"C2GS1"	M 2318.0	BOOL	// (C2RB.S4): GRUPO DE SEQUENCIA PESO 1
"C2GS2"	M 2318.1	BOOL	// (C2RB.S4): GRUPO DE SEQUENCIA PESO 2
"C2GS4"	M 2318.2	BOOL	// (C2RB.S4): GRUPO DE SEQUENCIA PESO 4
"C2GS8"	M 2318.3	BOOL	// (C2RB.S4): GRUPO DE SEQUENCIA PESO 8
"C2E1_SRE"	M 2318.4	BOOL	// (C2RB.S4): INFO DETECCION RETROCESOSEQUENCIA 1
"C2E1_SAV"	M 2318.5	BOOL	// (C2RB.S4): INFO DETECCION AVANCE SEQUENCIA 1
"C2E2_SRE"	M 2318.6	BOOL	// (C2RB.S4): INFO DETECCION RETROCESOSEQUENCIA 2
"C2E2_SAV"	M 2318.7	BOOL	// (C2RB.S4): INFO DETECCION AVANCE SEQUENCIA 2
"C2DECH"	M 2319.0	BOOL	// (C2RB.S4): COMANDE DESBLOQUEIO TROCADER
"C2EVO1"	M 2320.0	BOOL	// (C2RB.S5): EVENTO HERRAMIENTA 1
"C2EVO2"	M 2320.1	BOOL	// (C2RB.S5): EVENTO HERRAMIENTA 2
"C2EVO3"	M 2320.2	BOOL	// (C2RB.S5): EVENTO HERRAMIENTA 3
"C2EVO4"	M 2320.3	BOOL	// (C2RB.S5): EVENTO HERRAMIENTA 4
"C2EVO5"	M 2320.4	BOOL	// (C2RB.S5): EVENTO HERRAMIENTA 5
"C2EVO6"	M 2320.5	BOOL	// (C2RB.S5): EVENTO HERRAMIENTA 6
"C2EVO7"	M 2320.6	BOOL	// (C2RB.S5): EVENTO HERRAMIENTA 7
"C2EVO8"	M 2320.7	BOOL	// (C2RB.S5): EVENTO HERRAMIENTA 8
"C2EVO9"	M 2321.0	BOOL	// (C2RB.S5): EVENTO HERRAMIENTA 9
"C2EVO10"	M 2321.1	BOOL	// (C2RB.S5): EVENTO HERRAMIENTA 10
"C2EVO11"	M 2321.2	BOOL	// (C2RB.S5): EVENTO HERRAMIENTA 11
"C2EVO12"	M 2321.3	BOOL	// (C2RB.S5): EVENTO HERRAMIENTA 12
"C2EVO13"	M 2321.4	BOOL	// (C2RB.S5): EVENTO HERRAMIENTA 13
"C2EVO14"	M 2321.5	BOOL	// (C2RB.S5): EVENTO HERRAMIENTA 14
"C2EVO15"	M 2321.6	BOOL	// (C2RB.S5): EVENTO HERRAMIENTA 15
"C2EVO16"	M 2321.7	BOOL	// (C2RB.S5): EVENTO HERRAMIENTA 16
"C2EV17"	M 2326.0	BOOL	// (C2RB.S8): EVENTO 17
"C2EV18"	M 2326.1	BOOL	// (C2RB.S8): EVENTO 18
"C2EV19"	M 2326.2	BOOL	// (C2RB.S8): EVENTO 19
"C2EV20"	M 2326.3	BOOL	// (C2RB.S8): EVENTO 20
"C2EV21"	M 2326.4	BOOL	// (C2RB.S8): EVENTO 21
"C2EV22"	M 2326.5	BOOL	// (C2RB.S8): EVENTO 22
"C2EV23"	M 2326.6	BOOL	// (C2RB.S8): EVENTO 23
"C2EV24"	M 2326.7	BOOL	// (C2RB.S8): EVENTO 24
"C2EV25"	M 2327.0	BOOL	// (C2RB.S8): EVENTO 25
"C2EV26"	M 2327.1	BOOL	// (C2RB.S8): EVENTO 26
"C2EV27"	M 2327.2	BOOL	// (C2RB.S8): EVENTO 27
"C2EV28"	M 2327.3	BOOL	// (C2RB.S8): EVENTO 28
"C2EV29"	M 2327.4	BOOL	// (C2RB.S8): EVENTO 29
"C2EV30"	M 2327.5	BOOL	// (C2RB.S8): EVENTO 30
"C2EV31"	M 2327.6	BOOL	// (C2RB.S8): EVENTO 31
"C2EV32"	M 2327.7	BOOL	// (C2RB.S8): EVENTO 32
"A2RBMS1_P"	MB 2200	BYTE	// BYTE 1 GENERAL DATA / GENERALITES
"A2RBMS2_P"	MB 2201	BYTE	// BYTE 2 GENERAL DATA / GENERALITES
"A2RBMS3_P"	MB 2202	BYTE	// BYTE 3 ROBOTT ORDERS / ORDRES ROBOTT
"A2RBMS4_P"	MB 2203	BYTE	// BYTE 4 ROBOTT ORDERS / ORDRES ROBOTT
"A2RBMS5_P"	MB 2204	BYTE	// BYTE 5 GRIPPER AND TOOL CHANGER / PREHENSEUR ET CHANGEUR OUTIL
"A2RBMS6_P"	MB 2205	BYTE	// BYTE 6 GRIPPER AND TOOL CHANGER / PREHENSEUR ET CHANGEUR OUTIL
"A2RBMS7_P"	MB 2206	BYTE	// BYTE 7 FAULT NUMBER / NUMERO DE DEFAUT
"A2RBMS8_P"	MB 2207	BYTE	// BYTE 8 FAULT NUMBER / NUMERO DE DEFAUT
"A2RBMS9_P"	MB 2208	BYTE	// BYTE 9 TOOL ORDERS/ ORDRES OUTIL
"A2RBMS10_P"	MB 2209	BYTE	// BYTE 10 TOOL ORDERS/ ORDRES OUTIL
"A2RBMS11_P"	MB 2210	BYTE	// BYTE 11
"A2RBMS12_P"	MB 2211	BYTE	// BYTE 12
"A2RBMS13_P"	MB 2212	BYTE	// BYTE 13
"A2RBMS14_P"	MB 2213	BYTE	// BYTE 14
"A2RBMS15_P"	MB 2214	BYTE	// BYTE 15
"A2RBMS16_P"	MB 2215	BYTE	// BYTE 16
"A2RBME1_P"	MB 2216	BYTE	// BYTE 1 GENERAL DATA AND CYCLE CODE / CODE CYCLE ET GENERALITES
"A2RBME2_P"	MB 2217	BYTE	// BYTE 2 GENERAL DATA AND CYCLE CODE / CODE CYCLE ET GENERALITES
"A2RBME3_P"	MB 2218	BYTE	// BYTE 3 ROBOTT EVENTS / EVENTOS ROBOTT
"A2RBME4_P"	MB 2219	BYTE	// BYTE 4 ROBOTT EVENTS / EVENTOS ROBOTT
"A2RBME5_P"	MB 2220	BYTE	// BYTE 5 GENERAL DATAS / GENERALITES
"A2RBME6_P"	MB 2221	BYTE	// BYTE 6 GENERAL DATAS / GENERALITES
"A2RBME7_P"	MB 2222	BYTE	// BYTE 7 GRIPPER AND TOOL CHANGER / PREHENSEUR ET CHANGEUR OUTIL
"A2RBME8_P"	MB 2223	BYTE	// BYTE 8 GRIPPER AND TOOL CHANGER / PREHENSEUR ET CHANGEUR OUTIL
"A2RBME9_P"	MB 2224	BYTE	// BYTE 9 TOOL EVENTS / EVENTOS OUTIL
"A2RBME10_P"	MB 2225	BYTE	// BYTE 10 TOOL EVENTS / EVENTOS OUTIL
"A2RBME11_P"	MB 2226	BYTE	// BYTE 11
"A2RBME12_P"	MB 2227	BYTE	// BYTE 12
"A2RBME13_P"	MB 2228	BYTE	// BYTE 13
"A2RBME14_P"	MB 2229	BYTE	// BYTE 14
"A2RBME15_P"	MB 2230	BYTE	// BYTE 15
"A2RBME16_P"	MB 2231	BYTE	// BYTE 16
"A3RBMS1_P"	MB 2232	BYTE	// BYTE 1 GENERAL DATA / GENERALITES
"A3RBMS2_P"	MB 2233	BYTE	// BYTE 2 GENERAL DATA / GENERALITES
"A3RBMS3_P"	MB 2234	BYTE	// BYTE 3 ROBOTT ORDERS / ORDRES ROBOTT
"A3RBMS4_P"	MB 2235	BYTE	// BYTE 4 ROBOTT ORDERS / ORDRES ROBOTT
"A3RBMS5_P"	MB 2236	BYTE	// BYTE 5 GRIPPER AND TOOL CHANGER / PREHENSEUR ET CHANGEUR OUTIL
"A3RBMS6_P"	MB 2237	BYTE	// BYTE 6 GRIPPER AND TOOL CHANGER / PREHENSEUR ET CHANGEUR OUTIL
"A3RBMS7_P"	MB 2238	BYTE	// BYTE 7 FAULT NUMBER / NUMERO DE DEFAUT
"A3RBMS8_P"	MB 2239	BYTE	// BYTE 8 FAULT NUMBER / NUMERO DE DEFAUT
"A3RBMS9_P"	MB 2240	BYTE	// BYTE 9 TOOL ORDERS/ ORDRES OUTIL
"A3RBMS10_P"	MB 2241	BYTE	// BYTE 10 TOOL ORDERS/ ORDRES OUTIL
"A3RBMS11_P"	MB 2242	BYTE	// BYTE 11
"A3RBMS12_P"	MB 2243	BYTE	// BYTE 12
"A3RBMS13_P"	MB 2244	BYTE	// BYTE 13
"A3RBMS14_P"	MB 2245	BYTE	// BYTE 14
"A3RBMS15_P"	MB 2246	BYTE	// BYTE 15
"A3RBMS16_P"	MB 2247	BYTE	// BYTE 16
"A3RBME1_P"	MB 2248	BYTE	// BYTE 1 GENERAL DATA AND CYCLE CODE / CODE CYCLE ET GENERALITES
"A3RBME2_P"	MB 2249	BYTE	// BYTE 2 GENERAL DATA AND CYCLE CODE / CODE CYCLE ET GENERALITES
"A3RBME3_P"	MB 2250	BYTE	// BYTE 3 ROBOTT EVENTS / EVENTOS ROBOTT
"A3RBME4_P"	MB 2251	BYTE	// BYTE 4 ROBOTT EVENTS / EVENTOS ROBOTT
"A3RBME5_P"	MB 2252	BYTE	// BYTE 5 GENERAL DATAS / GENERALITES
"A3RBME6_P"	MB 2253	BYTE	// BYTE 6 GENERAL DATAS / GENERALITES
"A3RBME7_P"	MB 2254	BYTE	// BYTE 7 GRIPPER AND TOOL CHANGER / PREHENSEUR ET CHANGEUR OUTIL
"A3RBME8_P"	MB 2255	BYTE	// BYTE 8 GRIPPER AND TOOL CHANGER / PREHENSEUR ET CHANGEUR OUTIL
"A3RBME9_P"	MB 2256	BYTE	// BYTE 9 TOOL EVENTS / EVENTOS OUTIL
"A3RBME10_P"	MB 2257	BYTE	// BYTE 10 TOOL EVENTS / EVENTOS OUTIL
"A3RBME11_P"	MB 2258	BYTE	// BYTE 11
"A3RBME12_P"	MB 2259	BYTE	// BYTE 12
"A3RBME13_P"	MB 2260	BYTE	// BYTE 13
"A3RBME14_P"	MB 2261	BYTE	// BYTE 14
"A3RBME15_P"	MB 2262	BYTE	// BYTE 15
"A3RBME16_P"	MB 2263	BYTE	// BYTE 16
"C2RBMS1_P"	MB 2296	BYTE	// BYTE 1 GENERAL DATA / GENERALITES
"C2RBMS2_P"	MB 2297	BYTE	// BYTE 2 GENERAL DATA / GENERALITES
"C2RBMS3_P"	MB 2298	BYTE	// BYTE 3 ROBOTT ORDERS / ORDRES ROBOTT
"C2RBMS4_P"	MB 2299	BYTE	// BYTE 4 ROBOTT ORDERS / ORDRES ROBOTT
"C2RBMS5_P"	MB 2300	BYTE	// BYTE 5 GRIPPER AND TOOL CHANGER / PREHENSEUR ET CHANGEUR OUTIL
"C2RBMS6_P"	MB 2301	BYTE	// BYTE 6 GRIPPER AND TOOL CHANGER / PREHENSEUR ET CHANGEUR OUTIL
"C2RBMS7_P"	MB 2302	BYTE	// BYTE 7 FAULT NUMBER / NUMERO DE DEFAUT
"C2RBMS8_P"	MB 2303	BYTE	// BYTE 8 FAULT NUMBER / NUMERO DE DEFAUT
"C2RBMS9_P"	MB 2304	BYTE	// BYTE 9 TOOL ORDERS/ ORDRES OUTIL
"C2RBMS10_P"	MB 2305	BYTE	// BYTE 10 TOOL ORDERS/ ORDRES OUTIL
"C2RBMS11_P"	MB 2306	BYTE	// BYTE 11
"C2RBMS12_P"	MB 2307	BYTE	// BYTE 12
"C2RBMS13_P"	MB 2308	BYTE	// BYTE 13
"C2RBMS14_P"	MB 2309	BYTE	// BYTE 14
"C2RBMS15_P"	MB 2310	BYTE	// BYTE 15
"C2RBMS16_P"	MB 2311	BYTE	// BYTE 16
"C2RBME1_P"	MB 2312	BYTE	// BYTE 1 GENERAL DATA AND CYCLE CODE / CODE CYCLE ET GENERALITES
"C2RBME2_P"	MB 2313	BYTE	// BYTE 2 GENERAL DATA AND CYCLE CODE / CODE CYCLE ET GENERALITES
"C2RBME3_P"	MB 2314	BYTE	// BYTE 3 ROBOTT EVENTS / EVENTOS ROBOTT
"C2RBME4_P"	MB 2315	BYTE	// BYTE 4 ROBOTT EVENTS / EVENTOS ROBOTT
"C2RBME5_P"	MB 2316	BYTE	// BYTE 5 GENERAL DATAS / GENERALITES
"C2RBME6_P"	MB 2317	BYTE	// BYTE 6 GENERAL DATAS / GENERALITES
"C2RBME7_P"	MB 2318	BYTE	// BYTE 7 GRIPPER AND TOOL CHANGER / PREHENSEUR ET CHANGEUR OUTIL
"C2RBME8_P"	MB 2319	BYTE	// BYTE 8 GRIPPER AND TOOL CHANGER / PREHENSEUR ET CHANGEUR OUTIL
"C2RBME9_P"	MB 2320	BYTE	// BYTE 9 TOOL EVENTS / EVENTOS OUTIL
"C2RBME10_P"	MB 2321	BYTE	// BYTE 10 TOOL EVENTS / EVENTOS OUTIL
"C2RBME11_P"	MB 2322	BYTE	// BYTE 11
"C2RBME12_P"	MB 2323	BYTE	// BYTE 12
"C2RBME13_P"	MB 2324	BYTE	// BYTE 13
"C2RBME14_P"	MB 2325	BYTE	// BYTE 14
"C2RBME15_P"	MB 2326	BYTE	// BYTE 15
"C2RBME16_P"	MB 2327	BYTE	// BYTE 16
"A2RBMS1_W"	MW 2200	WORD	// WORD 1 GENERAL DATA / GENERALITES
"A2RBMS2_W"	MW 2202	WORD	// WORD 2 ROBOTT ORDERS / ORDRES ROBOTT
"A2RBMS3_W"	MW 2204	WORD	// WORD 3 GRIPPER AND TOOL CHANGER / PREHENSEUR ET CHANGEUR OUTIL
"A2RBMS4_W"	MW 2206	WORD	// WORD 4 FAULT NUMBER / NUMERO DE DEFAUT
"A2RBMS5_W"	MW 2208	WORD	// WORD 5 TOOL ORDERS/ ORDRES OUTIL
"A2RBMS6_W"	MW 2210	WORD	// WORD 6
"A2RBMS7_W"	MW 2212	WORD	// WORD 7
"A2RBMS8_W"	MW 2214	WORD	// WORD 8
"A2RBME1_W"	MW 2216	WORD	// WORD 1 GENERAL DATA AND CYCLE CODE / CODE CYCLE ET GENERALITES
"A2RBME2_W"	MW 2218	WORD	// WORD 2 ROBOTT EVENTS / EVENTOS ROBOTT
"A2RBME3_W"	MW 2220	WORD	// WORD 3 GENERAL DATAS / GENERALITES
"A2RBME4_W"	MW 2222	WORD	// WORD 4 GRIPPER AND TOOL CHANGER / PREHENSEUR ET CHANGEUR OUTIL
"A2RBME5_W"	MW 2224	WORD	// WORD 5 TOOL EVENTS / EVENTOS OUTIL
"A2RBME6_W"	MW 2226	WORD	// WORD 6
"A2RBME7_W"	MW 2228	WORD	// WORD 7
"A2RBME8_W"	MW 2230	WORD	// WORD 8
"A3RBMS1_W"	MW 2232	WORD	// WORD 1 GENERAL DATA / GENERALITES
"A3RBMS2_W"	MW 2234	WORD	// WORD 2 ROBOTT ORDERS / ORDRES ROBOTT
"A3RBMS3_W"	MW 2236	WORD	// WORD 3 GRIPPER AND TOOL CHANGER / PREHENSEUR ET CHANGEUR OUTIL
"A3RBMS4_W"	MW 2238	WORD	// WORD 4 FAULT NUMWER / NUMERO DE DEFAUT
"A3RBMS5_W"	MW 2240	WORD	// WORD 5 TOOL ORDERS/ ORDRES OUTIL
"A3RBMS6_W"	MW 2242	WORD	// WORD 6
"A3RBMS7_W"	MW 2244	WORD	// WORD 7
"A3RBMS8_W"	MW 2246	WORD	// WORD 8
"A3RBME1_W"	MW 2248	WORD	// WORD 1 GENERAL DATA AND CYCLE CODE / CODE CYCLE ET GENERALITES
"A3RBME2_W"	MW 2250	WORD	// WORD 2 ROBOTT EVENTS / EVENTOS ROBOTT
"A3RBME3_W"	MW 2252	WORD	// WORD 3 GENERAL DATAS / GENERALITES
"A3RBME4_W"	MW 2254	WORD	// WORD 4 GRIPPER AND TOOL CHANGER / PREHENSEUR ET CHANGEUR OUTIL
"A3RBME5_W"	MW 2256	WORD	// WORD 5 TOOL EVENTS / EVENTOS OUTIL
"A3RBME6_W"	MW 2258	WORD	// WORD 6
"A3RBME7_W"	MW 2260	WORD	// WORD 7
"A3RBME8_W"	MW 2262	WORD	// WORD 8
"C2RBMS1_W"	MW 2296	WORD	// WORD 1 GENERAL DATA / GENERALITES
"C2RBMS2_W"	MW 2298	WORD	// WORD 2 ROBOTT ORDERS / ORDRES ROBOTT
"C2RBMS3_W"	MW 2300	WORD	// WORD 3 GRIPPER AND TOOL CHANGER / PREHENSEUR ET CHANGEUR OUTIL
"C2RBMS4_W"	MW 2302	WORD	// WORD 4 FAULT NUMWER / NUMERO DE DEFAUT
"C2RBMS5_W"	MW 2304	WORD	// WORD 5 TOOL ORDERS/ ORDRES OUTIL
"C2RBMS6_W"	MW 2306	WORD	// WORD 6
"C2RBMS7_W"	MW 2308	WORD	// WORD 7
"C2RBMS8_W"	MW 2310	WORD	// WORD 8
"C2RBME1_W"	MW 2312	WORD	// WORD 1 GENERAL DATA AND CYCLE CODE / CODE CYCLE ET GENERALITES
"C2RBME2_W"	MW 2314	WORD	// WORD 2 ROBOTT EVENTS / EVENTOS ROBOTT
"C2RBME3_W"	MW 2316	WORD	// WORD 3 GENERAL DATAS / GENERALITES
"C2RBME4_W"	MW 2318	WORD	// WORD 4 GRIPPER AND TOOL CHANGER / PREHENSEUR ET CHANGEUR OUTIL
"C2RBME5_W"	MW 2320	WORD	// WORD 5 TOOL EVENTS / EVENTOS OUTIL
"C2RBME6_W"	MW 2322	WORD	// WORD 6
"C2RBME7_W"	MW 2324	WORD	// WORD 7
"C2RBME8_W"	MW 2326	WORD	// WORD 8
"CYCL_EXC"	OB 1	OB 1	// EXECUTION CYCLE
"CYC_INT4"	OB 34	OB 34	// CYCLIC INTERRUPT 4
"CYCL_FLT"	OB 80	OB 80	// Cycle Time Fault
"I/O_FLT1"	OB 82	OB 82	// I/O POINT FAULT 1
"I/O_FLT2"	OB 83	OB 83	// I/O POINT FAULT 2
"OBNL_FLT"	OB 85	OB 85	// OB NOT LOADED FAULT
"RACK_FLT"	OB 86	OB 86	// LOSS OF RACK FAULT
"COMPLETE RESTART"	OB 100	OB 100	// COMPLETE RESTART
"PROG_ERR"	OB 121	OB 121	// Programming Error
"MOD_ERR"	OB 122	OB 122	// MODULE ACCESS ERROR
"VADI"	Q 0.0	BOOL	// (MOP-IM.M06-07): INDICDOR RESET FALLA
"VMCY"	Q 0.1	BOOL	// (MOP-IM.M06-07): INDICADOR MARCHA CICLO
"VAOP"	Q 0.3	BOOL	// (MOP-IM.M06-07): ALIMENTADOR APPEL OPERADOR
"Z1VROC"	Q 10.0	BOOL	// (Z1ZB.M05): INDICADOR Retorno Origen
"Z1RCM"	Q 10.7	BOOL	// (Z1ZB.M05): RELE DE CONTROL DE MASA
"RAU"	Q 25.0	BOOL	// (Z1ZB.M15): RELE COMUN DE SEGURIDAD SC1 (Z1AU)
"RES"	Q 25.1	BOOL	// (Z1ZB.M15): RELE COMUN DE SEGURIDAD ES
"RFZ"	Q 25.2	BOOL	// (Z1ZB.M15): RELE COMUN DE SEGURIDAD FZ
"RSC4"	Q 25.3	BOOL	// (Z1ZB.M15): RELE COMUN DE SEGURIDAD RL
"WB11"	Q 42.0	BOOL	// (Z1ZB.M08):Welding Box 1 Bit 1
"WB12"	Q 42.1	BOOL	// (Z1ZB.M08):Welding Box 1 Bit 2
"WB13"	Q 42.2	BOOL	// (Z1ZB.M08):Welding Box 1 Bit 3
"WB14"	Q 42.3	BOOL	// (Z1ZB.M08):Welding Box 1 Bit 4
"WB21"	Q 42.4	BOOL	// (Z1ZB.M08):Welding Box 2 Bit 1
"WB22"	Q 42.5	BOOL	// (Z1ZB.M08):Welding Box 2 Bit 2
"WB23"	Q 42.6	BOOL	// (Z1ZB.M08):Welding Box 2 Bit 3
"WB24"	Q 42.7	BOOL	// (Z1ZB.M08):Welding Box 2 Bit 4
"OP1VAT"	Q 43.0	BOOL	// (Z1ZB.M09): Work Autorisation Lamp 1 (Green)
"OP1VIT"	Q 43.1	BOOL	// (Z1ZB.M09): Work Prohibition Lamp 1 (Red)
"OP1VDF"	Q 43.2	BOOL	// (Z1ZB.M09): Default Lamp 1 (Orange)
"A0CBNOK"	Q 43.3	BOOL	// (Z1ZB.M09): BARCODE READING NOK
"A0CBOK"	Q 43.4	BOOL	// (Z1ZB.M09): BARCODE READING OK
"OP2VAT"	Q 43.5	BOOL	// (Z1ZB.M09): Work Autorisation Lamp 2 (Green)
"OP2VIT"	Q 43.6	BOOL	// (Z1ZB.M09): Work Prohibition Lamp 2 (Red)
"OP2VDF"	Q 43.7	BOOL	// (Z1ZB.M09): Default Lamp 2 (Orange)
"A0EACH1"	Q 60.0	BOOL	// ELECTROVALVE AV CH1
"A0ERCH1"	Q 60.1	BOOL	// ELECTROVALVE RET CH1
"A0EAVR2"	Q 60.2	BOOL	// ELECTROVALVE AV VR2
"A0ERVR2"	Q 60.3	BOOL	// ELECTROVALVE RET VR2
"A0EAVR3"	Q 60.4	BOOL	// ELECTROVALVE AV VR3
"A0ERVR3"	Q 60.5	BOOL	// ELECTROVALVE RET VR3
"A0EASR4"	Q 60.6	BOOL	// ELECTROVALVE AV SR4
"A0ERSR4"	Q 60.7	BOOL	// ELECTROVALVE RET SR4
"A0EASR5"	Q 61.0	BOOL	// ELECTROVALVE AV SR5
"A0ERSR5"	Q 61.1	BOOL	// ELECTROVALVE RET SR5
"A0EASR6"	Q 61.2	BOOL	// ELECTROVALVE AV SR6
"A0ERSR6"	Q 61.3	BOOL	// ELECTROVALVE RET SR6
"A0EASR7"	Q 61.4	BOOL	// ELECTROVALVE AV SR7
"A0ERSR7"	Q 61.5	BOOL	// ELECTROVALVE RET SR7
"A0EASR9"	Q 62.0	BOOL	// ELECTROVALVE AV SR9
"A0ERSR9"	Q 62.1	BOOL	// ELECTROVALVE RET SR9
"A0RSOP"	Q 68.0	BOOL	// (A0IM1-FVD0): SEG OPERADOR
"A0EV"	Q 68.2	BOOL	// (A0IM1-FVD0): PILOTAGE ELETROVALVE (COMMON ES)
"A0_DO8"	Q 259.0	BOOL	// (A0SBS120): DIGITAL OUTPUT 8
"A0_DO9"	Q 259.1	BOOL	// (A0SBS120): DIGITAL OUTPUT 9
"A0_DO10"	Q 259.2	BOOL	// (A0SBS120): DIGITAL OUTPUT 10
"A0_DO11"	Q 259.3	BOOL	// (A0SBS120): DIGITAL OUTPUT 11
"A0_STO_O"	Q 312.0	BOOL	// (A0SBS120): ENABLE STO
"A0_SS1_O"	Q 312.1	BOOL	// (A0SBS120): ENABLE SS1
"A0_SS2_O"	Q 312.2	BOOL	// (A0SBS120): ENABLE SS2
"A0_SOS_O"	Q 312.3	BOOL	// (A0SBS120): ENABLE SOS
"A0_SLS_O"	Q 312.4	BOOL	// (A0SBS120): ENABLE SLS
"A0_RES1_O"	Q 312.5	BOOL	// (A0SBS120): RESERVE
"A0_RES2_O"	Q 312.6	BOOL	// (A0SBS120): RESERVE
"A0_ACK_O"	Q 312.7	BOOL	// (A0SBS120): ACK
"A0_RES3_O"	Q 313.0	BOOL	// (A0SBS120): RESERVE
"A0_L1SLS_O"	Q 313.1	BOOL	// (A0SBS120): ENABLE LIMIT 1 SLS
"A0_L2SLS_O"	Q 313.2	BOOL	// (A0SBS120): ENABLE LIMIT 2 SLS
"A0_RES4_O"	Q 313.3	BOOL	// (A0SBS120): RESERVE
"A0_RES5_O"	Q 313.4	BOOL	// (A0SBS120): RESERVE
"A0_RES6_O"	Q 313.5	BOOL	// (A0SBS120): RESERVE
"A0_RES7_O"	Q 313.6	BOOL	// (A0SBS120): RESERVE
"A0_RES8_O"	Q 313.7	BOOL	// (A0SBS120): RESERVE
"Z1SPA1VMCY"	Q 350.7	BOOL	// (Z1SPA1.O0): INDICADOR MARCHA CICLO
"Z1SPA1VDACY"	Q 351.0	BOOL	// (Z1SPA1.O1): INDICADOR DEMANDA PARADA CICLO
"Z2VROC"	Q 400.0	BOOL	// (Z2ZB.M07): INDICADOR Retorno Origen
"Z2VMCY"	Q 400.1	BOOL	// Z2ZB[M07]: LAMP CYCLE RUN (SOP)
"Z2RCM"	Q 400.7	BOOL	// (Z2ZB.M07): RELE DE CONTROL DE MASA
"B0WB11"	Q 401.0	BOOL	// (Z2ZB.M08):Welding Box 1 Bit 1
"B0WB12"	Q 401.1	BOOL	// (Z2ZB.M08):Welding Box 1 Bit 2
"B0WB13"	Q 401.2	BOOL	// (Z2ZB.M08):Welding Box 1 Bit 3
"B0WB14"	Q 401.3	BOOL	// (Z2ZB.M08):Welding Box 1 Bit 4
"B0WB21"	Q 401.4	BOOL	// (Z2ZB.M08):Welding Box 2 Bit 1
"B0WB22"	Q 401.5	BOOL	// (Z2ZB.M08):Welding Box 2 Bit 2
"B0WB23"	Q 401.6	BOOL	// (Z2ZB.M08):Welding Box 2 Bit 3
"B0WB24"	Q 401.7	BOOL	// (Z2ZB.M08):Welding Box 2 Bit 4
"B0OP1VAT"	Q 402.0	BOOL	// (Z2ZB.M08): Work Autorisation Lamp 1 (Green)
"B0OP1VIT"	Q 402.1	BOOL	// (Z2ZB.M08): Work Prohibition Lamp 1 (Red)
"B0OP1VDF"	Q 402.2	BOOL	// (Z2ZB.M08): Default Lamp 1 (Orange)
"A402.3"	Q 402.3	BOOL	// (Z2ZB.M08): RESERVE
"A402.4"	Q 402.4	BOOL	// (Z2ZB.M08): RESERVE
"B0OP2VAT"	Q 402.5	BOOL	// (Z2ZB.M08): Work Autorisation Lamp 2 (Green)
"B0OP2VIT"	Q 402.6	BOOL	// (Z2ZB.M08): Work Prohibition Lamp 2 (Red)
"B0OP2VDF"	Q 402.7	BOOL	// (Z2ZB.M08): Default Lamp 2 (Orange)
"B0RAU"	Q 423.0	BOOL	// (Z2ZB.M13): RELE COMUN DE SEGURIDAD SC1 (Z2AU)
"B0RES"	Q 423.1	BOOL	// (Z2ZB.M13): RELE COMUN DE SEGURIDAD ES
"B0RFZ"	Q 423.2	BOOL	// (Z2ZB.M13): RELE COMUN DE SEGURIDAD FZ
"B0RSC4"	Q 423.3	BOOL	// (Z2ZB.M13): RELE COMUN DE SOP
"B0EASR1"	Q 450.0	BOOL	// ELECTROVALVE AV SR1
"B0ERSR1"	Q 450.1	BOOL	// ELECTROVALVE RET SR1
"B0EASR2"	Q 450.2	BOOL	// ELECTROVALVE AV SR2
"B0ERSR2"	Q 450.3	BOOL	// ELECTROVALVE RET SR2
"B0EASR3"	Q 450.4	BOOL	// ELECTROVALVE AV SR3
"B0ERSR3"	Q 450.5	BOOL	// ELECTROVALVE RET SR3
"B0EASR4"	Q 450.6	BOOL	// ELECTROVALVE AV SR4
"B0ERSR4"	Q 450.7	BOOL	// ELECTROVALVE RET SR4
"B0EASR5"	Q 451.0	BOOL	// ELECTROVALVE AV SR5
"B0ERSR5"	Q 451.1	BOOL	// ELECTROVALVE RET SR5
"B0EASR6"	Q 451.2	BOOL	// ELECTROVALVE AV SR6
"B0ERSR6"	Q 451.3	BOOL	// ELECTROVALVE RET SR6
"B0EASR7"	Q 451.4	BOOL	// ELECTROVALVE AV SR7
"B0ERSR7"	Q 451.5	BOOL	// ELECTROVALVE RET SR7
"B0EASR8"	Q 451.6	BOOL	// ELECTROVALVE AV SR8
"B0ERSR8"	Q 451.7	BOOL	// ELECTROVALVE RET SR8
"B0EACL9"	Q 452.0	BOOL	// ELECTROVALVE AV CL9
"B0ERCL9"	Q 452.1	BOOL	// ELECTROVALVE RET CL9
"B0EACL10"	Q 452.2	BOOL	// ELECTROVALVE AV CL10
"B0ERCL10"	Q 452.3	BOOL	// ELECTROVALVE RET CL10
"RES1"	Q 452.4	BOOL
"RES2"	Q 452.5	BOOL
"RES3"	Q 452.6	BOOL
"RES4"	Q 452.7	BOOL
"Z2SPA1VMCY"	Q 490.7	BOOL	// (Z2SPA1.O0): INDICADOR MARCHA CICLO
"Z2SPA1VDACY"	Q 491.0	BOOL	// (Z2SPA1.O1): INDICADOR DEMANDA PARADA CICLO
"BOSEW_POS_ESCRITA"	QW 434	WORD
"TP"	SFB 3	SFB 3	// GENERATE A PULSE
"TON"	SFB 4	SFB 4	// GENERATE AN ON DELAY
"TOF"	SFB 5	SFB 5	// GENERATE AN OFF DELAY
"RDREC"	SFB 52	SFB 52	// READ A PROCESS DATA RECORD
"WRREC"	SFB 53	SFB 53	// WRITE A PROCESS DATA RECORD
"RALRM"	SFB 54	SFB 54	// Receive Alarm Data
"SET_CLK"	SFC 0	SFC 0	// SET SYSTEM CLOCK
"READ_CLK"	SFC 1	SFC 1	// READ SYSTEM CLOCK
"RD_SINFO"	SFC 6	SFC 6	// READ OB START INFORMATION
"D_ACT_DP"	SFC 12	SFC 12	// DEACTIVATING AND ACTIVATING DP SLAVES
"DPRD_DAT"	SFC 14	SFC 14	// READ CONSISTENT DATA OF A STANDARD DP SLAVE
"DPWR_DAT"	SFC 15	SFC 15	// WRITE CONSISTENT DATA TO A STANDARD DP SLAVE
"ALARM_SQ"	SFC 17	SFC 17	// Generate Block-Related Messages with Acknowledgment
"BLKMOV"	SFC 20	SFC 20	// COPY VARIABLES
"FILL"	SFC 21	SFC 21	// INITIALIZE A MEMORY AREA
"TEST_DB"	SFC 24	SFC 24	// TEST DATA BLOCK
"DIS_AIRT"	SFC 41	SFC 41	// DELAY THE HIGHER PRIORITY INTERRUPTS AND ASYNCHRONOUS ERRORS
"EN_AIRT"	SFC 42	SFC 42	// ENABLE HIGHER PRIORITY INTERRUPTS AND ASYNCHRONOUS ERRORS
"STP"	SFC 46	SFC 46	// CHANGE THE CPU TO STOP
"RDSYSST"	SFC 51	SFC 51	// READ A SYSTEM STATUS LIST OR PARTIAL LIST
"WR_REC"	SFC 58	SFC 58	// WRITE DATA RECORD
"RD_REC"	SFC 59	SFC 59	// READ A DATA RECORD
"TIME_TCK"	SFC 64	SFC 64	// READ THE SYSTEM TIME
"GEO_LOG"	SFC 70	SFC 70	// DETERMINE LOGICAL ADDRESS
"READ_DBL"	SFC 83	SFC 83	// READ DATA BLOCK OUT OF LOAD MEMORY
"WRIT_DBL"	SFC 84	SFC 84	// WRITE DATA BLOCK IN LOAD MEMORY
"DEL_SI"	SFC 106	SFC 106	// Deleting Dynamically Assigned System Instances
"ALARM_DQ"	SFC 107	SFC 107	// Creating Acknowledgeable Block-related Message
"ALARM_D"	SFC 108	SFC 108	// Creating Acknowledged Block-related Message
"MOT_FONC_NC"	UDT 1827	UDT 1827	// UDT utilisée en entrée des BF locator
"LIEN_PUP"	UDT 1988	UDT 1988	// Gestion des Modes et des pupitres de cde manu de la  zone (BF_ZONE_MODE_IHM)
"LIEN_ILOT"	UDT 2004	UDT 2004	// INFO CONTROL LINKED TO THE FACILITY (BF_ILOT)
"MOT_FONC_MP"	UDT 2041	UDT 2041	// INFO CONTROL OF A MOVEMENT (BF_MOUVMP1)
"MOT_FONC"	UDT 2042	UDT 2042	// INFO D'UN MOUVEMENT (BF_MOUV2P1,BF_MVSE2P1, BF_RB_COD_PREH_API)
"VAT_1"	VAT 1	
"VAT_cpx"	VAT 2	
"VAT_CPX_A02"	VAT 3	
"VARIADOR"	VAT 4	
"Prueba_N"	VAT 5	
"posiciones"	VAT 6	
"SEW"	VAT 7	
"Forzar"	VAT 8	
"B0_CAB"	VAT 9	
END_SYMBOL_TABLE
